PROGRAM interlocks
VAR PERSISTENT
	nv_3110_open: BOOL;
	alm_lt_3012_low: BOOL;
	intlk_u3112: BOOL;
	nv_3210_open: BOOL;
	nv_3310_open: BOOL;
	intlk_u3212: BOOL;
	intlk_u3312: BOOL;
	alm_lt_3102_low: BOOL;
	alm_lt_3202_low: BOOL;
	alm_lt_3302_low: BOOL;
	alm_lt_3153_low: BOOL;
	intlk_u3160: BOOL;
	alm_lt_3253_low: BOOL;
	intlk_u3260: BOOL;
	alm_lt_3353_low: BOOL;
	intlk_u3360: BOOL;
	nv_3372_open: BOOL;
	intlk_u3370: BOOL;
	alm_lt_3402_low: BOOL;
	nv_3135_open: BOOL;
	nv_3235_open: BOOL;
	nv_3335: BOOL;
	nv_3335_open: BOOL;
	intlk_nv3110: BOOL;
	u_3112_running: BOOL;
END_VAR

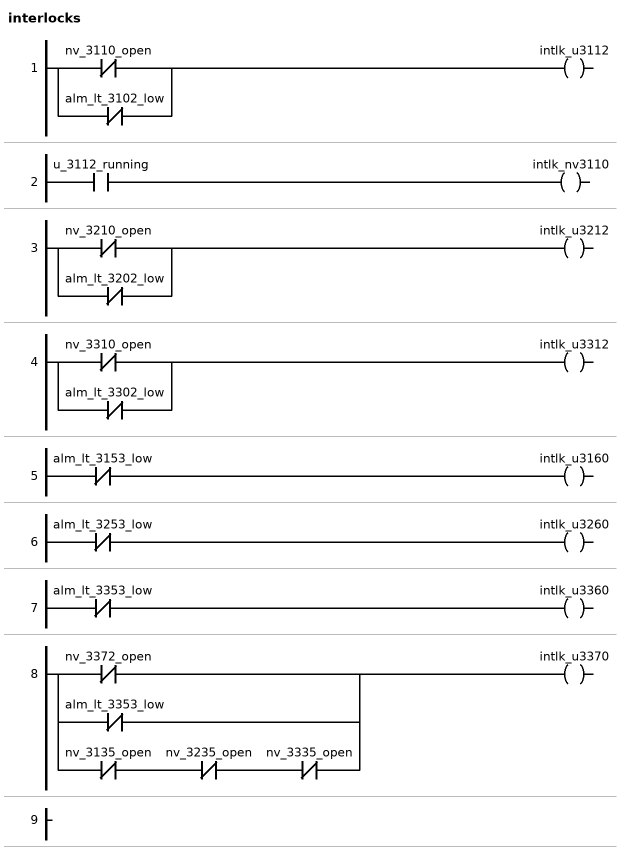
// NETWORK 1
intlk_u3112 := NOT nv_3110_open OR NOT alm_lt_3102_low;

// NETWORK 2
intlk_nv3110 := u_3112_running;

// NETWORK 3
intlk_u3212 := NOT nv_3210_open OR NOT alm_lt_3202_low;

// NETWORK 4
intlk_u3312 := NOT nv_3310_open OR NOT alm_lt_3302_low;

// NETWORK 5
intlk_u3160 := NOT alm_lt_3153_low;

// NETWORK 6
intlk_u3260 := NOT alm_lt_3253_low;

// NETWORK 7
intlk_u3360 := NOT alm_lt_3353_low;

// NETWORK 8
intlk_u3370 := NOT nv_3372_open OR NOT alm_lt_3353_low OR NOT nv_3135_open AND NOT nv_3235_open AND NOT nv_3335_open;

// NETWORK 9

END_PROGRAM

(* stored: Version 1.1.0.1, ProductVersion 3.1.4024.12
   POU interlocks: Id {5e6ac187-5fbb-479f-b495-0ce9f8a80e37}, SpecialFunc None *)
